FUNCTION_BLOCK Queue IMPLEMENTS I_Station, I_Cyclic, I_Resettable, I_Object
VAR
	_Position : LREAL := 0.0;
	_MyMover : I_XtsMover;
	_MyLeavingMover : I_XtsMover;
	_NullMover : I_XtsMover;
	_MyStation : I_Station;
	QueueSequence : INT;
	_isComplete : BOOL;
END_VAR

METHOD Cycle : HRESULT
CASE QueueSequence OF
	0:
		IF _MyMover <> 0 AND _MyStation.IsReady() THEN
			_MyLeavingMover := _MyMover;
			_MyMover := 0;
			_isComplete := TRUE;
			QueueSequence := 10;
		END_IF
	10:
		_isComplete := FALSE;
		IF _MyStation.IsOperating() THEN
			_MyLeavingMover := _NullMover;
			QueueSequence := 0;
		END_IF
END_CASE
END_METHOD

//FB_Init is always available implicitly and it is used primarily for initialization.
//The return value is not evaluated. For a specific influence, you can also declare the
//methods explicitly and provide additional code there with the standard initialization
//code. You can evaluate the return value.
METHOD FB_Init: BOOL
VAR_INPUT
    bInitRetains: BOOL; // TRUE: the retain variables are initialized (reset warm / reset cold)
    bInCopyCode: BOOL;  // TRUE: the instance will be copied to the copy code afterward (online change)  
	Position : LREAL; 
	Station : I_Station;
END_VAR
_Position := Position;
_MyStation := Station;
END_METHOD

METHOD HasMover : BOOL
HasMover := _MyMover <> 0;
END_METHOD

METHOD IsClear : BOOL
IsClear := _MyMover = 0;
END_METHOD

METHOD isComplete : BOOL
isComplete := _isComplete;
END_METHOD

METHOD IsOperating : BOOL
IsOperating := _MyMover <> 0;
END_METHOD

METHOD IsReady : BOOL
END_METHOD

METHOD MyMover : HRESULT
VAR_INPUT
	mover	: I_XtsMover;
END_VAR
IF mover = 0 THEN
	MyMover := -1;
	RETURN;
END_IF
IF _MyMover <> 0 THEN
	MyMover := -2;
	RETURN;
END_IF
_MyMover := mover;
END_METHOD

PROPERTY Position : MC_LREAL
GET
Position := _Position;
END_GET
END_PROPERTY

METHOD RegisterWithParent
VAR_INPUT
	Parent	: I_HostObjects;
END_VAR
END_METHOD

METHOD Reset : HRESULT
_isComplete := FALSE;
QueueSequence := 0;
END_METHOD

END_FUNCTION_BLOCK

(* stored: Version 1.1.0.1
   POU Queue: Id {8254c78a-3a7c-4581-9f3c-a41ac2249f11}, SpecialFunc None
   Folder Status: Id {4146ad9b-933c-4afb-a6d8-e90fa8366732}
   Method Cycle: Id {b03e5178-a63f-46c3-93a2-0179449aa637}
   Method FB_Init: Id {4a31526b-83cb-4557-8684-f1f086ebc0fe}
   Method HasMover: Id {20126ae5-2a64-4e3a-8bf1-40f04bba8f58}
   Method IsClear: Id {aed4f67a-12c4-44b3-89bd-dc10f74faa45}
   Method isComplete: Id {e755abc1-1f3a-493a-ad81-ab0e742a23ce}
   Method IsOperating: Id {f8703c69-d9e6-477e-882a-a6573d8c661c}
   Method IsReady: Id {6c981551-1b51-4198-93c9-7e75e7c31277}
   Method MyMover: Id {0c3e317f-08a9-475b-b84d-7ac86f2701cd}
   Property Position: Id {0fc938c1-886d-4378-832a-c7a96a3aba48}
   Get Get: Id {f1f2b796-050a-4f8f-ab96-64accc9dc6d5}
   Method RegisterWithParent: Id {e4dbf09d-b223-4b91-aece-dfac327a7503}
   Method Reset: Id {145e41f3-13a0-4491-94e4-c131fa0d6b67} *)
